(* PLC project Unnamed, Unknown Unnamed 1 *)
(* stored: creationDateTime 2025-08-19T02:55:19, modificationDateTime 2025-08-19T03:30:57 *)

PROGRAM program0
  VAR
    staff1 : BOOL;
    staff2 : BOOL;
    bio1 : BOOL;
    bio2 : BOOL;
    bio3 : BOOL;
    HEAD : BOOL;
    DOOR_OPEN : BOOL;
    stop : BOOL;
    start : BOOL;
    safety1 : BOOL;
    safety2 : BOOL;
    safety3 : BOOL;
    no_fault : BOOL;
    machine1 : BOOL;
    machine2 : BOOL;
    machine3 : BOOL;
    condition1 : BOOL;
    condition2 : BOOL;
    output : BOOL;
    main_valve : BOOL;
    level_sensor : BOOL;
    no_leak : BOOL;
    s1 : BOOL;
    s2 : BOOL;
    tank_OPEN : BOOL;
    P1 : BOOL;
    P2 : BOOL;
    output1 : BOOL;
    robotic_arm : BOOL;
  END_VAR

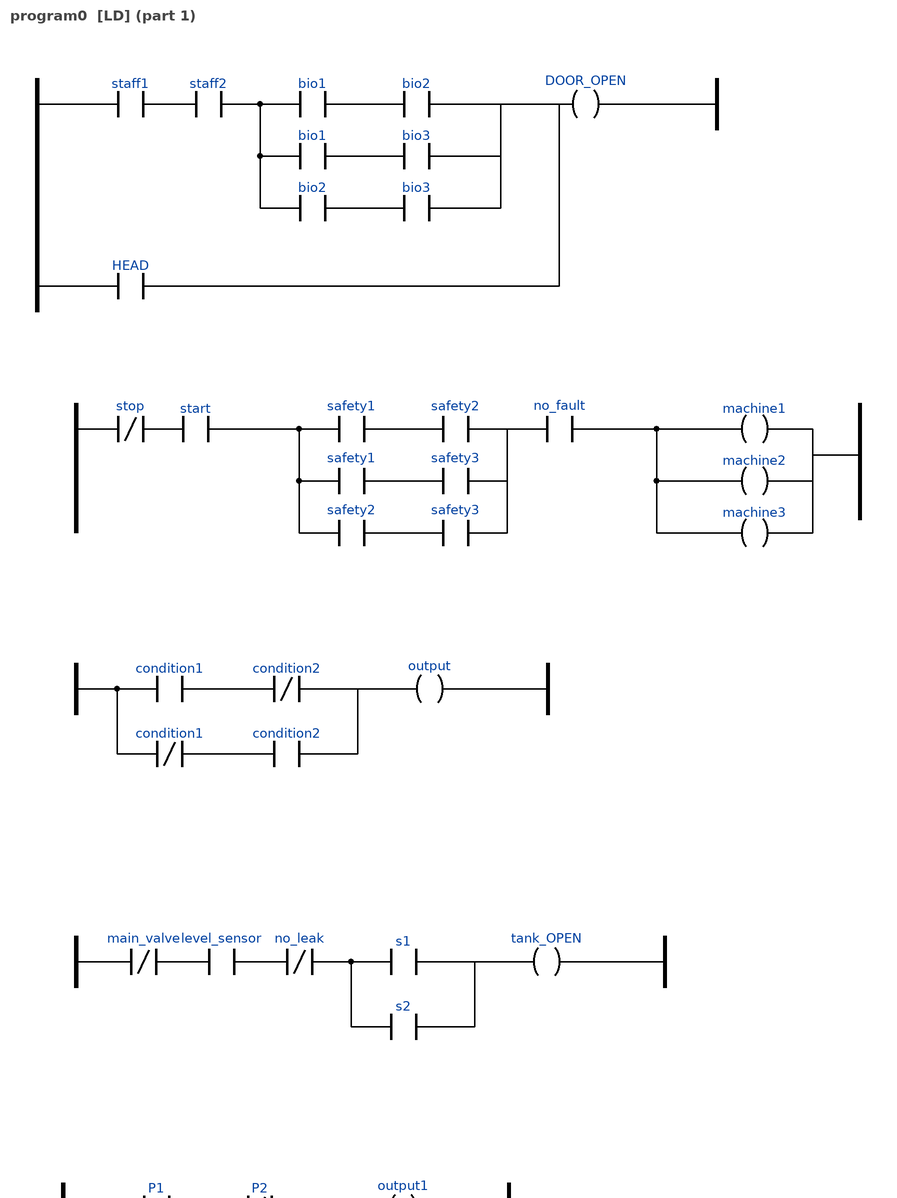
(* LD diagram, written out as Structured Text *)
DOOR_OPEN := staff1 AND staff2 AND bio1 AND bio2 OR staff1 AND staff2 AND bio1 AND bio3 OR staff1 AND staff2 AND bio2 AND bio3 OR HEAD;
machine1 := NOT stop AND start AND (safety1 AND safety2 OR safety1 AND safety3 OR safety2 AND safety3) AND no_fault;
machine2 := NOT stop AND start AND (safety1 AND safety2 OR safety1 AND safety3 OR safety2 AND safety3) AND no_fault;
machine3 := NOT stop AND start AND (safety1 AND safety2 OR safety1 AND safety3 OR safety2 AND safety3) AND no_fault;
output := condition1 AND NOT condition2 OR NOT condition1 AND condition2;
tank_OPEN := NOT main_valve AND level_sensor AND NOT no_leak AND (s2 OR s1);
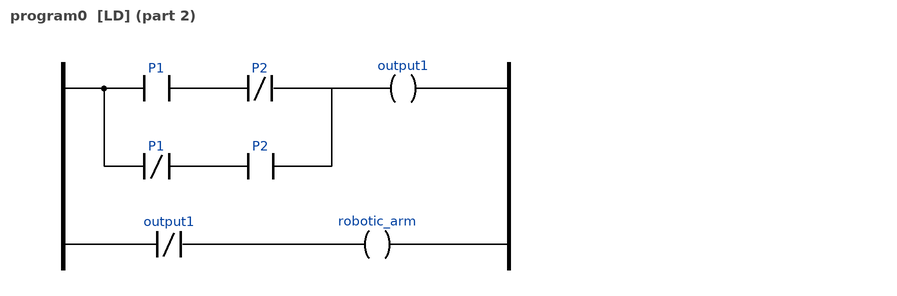
output1 := NOT P1 AND P2 OR P1 AND NOT P2;
robotic_arm := NOT output1;
END_PROGRAM

CONFIGURATION Config0
  RESOURCE Res0 ON PLC
    TASK task0(INTERVAL := T#20ms, PRIORITY := 0);
    PROGRAM instance0 WITH task0 : program0;
  END_RESOURCE
END_CONFIGURATION
